TYPE ST_SubStructure :
STRUCT
	e : LREAL;
	f : DT;
END_STRUCT
END_TYPE

(* stored: Version 1.1.0.1, ProductVersion 3.1.4022.12
   DUT ST_SubStructure: Id {95c86f74-48d4-4939-9ca3-8e07c63ef268} *)
